(* IEC 61131-3 sources: generating_plc_code_with_llms/Code#2/ChatGPT_3.5/third run, 21 files *)

(* ---- 14.st ---- *)
// 7.98s
// 2
FUNCTION FC1001 : BOOL
VAR_INPUT
	MEW: REAL;
	SP: REAL;
	HYS: REAL;
END_VAR

VAR_IN_OUT
 	OUT: BOOL;
END_VAR

VAR
 	P_HYS: REAL;
END_VAR

// Calculate the switching hysteresis value
P_HYS := SP * (HYS / 100.0);

// Switch on if the measured value exceeds the setpoint + hysteresis
IF MEW > (SP + P_HYS) THEN
    OUT := TRUE;
END_IF;

// Switch off if the measured value falls below the setpoint - hysteresis
IF MEW < (SP - P_HYS) THEN
    OUT := FALSE;
END_IF;

// Return the output state
RETURN OUT;

END_FUNCTION

(* ---- 15.st ---- *)
// 11.59s
// 2
FUNCTION FC1002 : BOOL
VAR_INPUT
	E_A, SENSOR: BOOL;
	ZEITW: TIME;
END_VAR

VAR_IN_OUT
	ZEIT: TON;
	P_HU, P_AL: BOOL;
END_VAR

// Check if the monitoring system is switched on
IF E_A THEN
    // Check if the ultrasonic sensor detects an approach
    IF SENSOR THEN
        // Start the timer if it's not running
        IF NOT ZEIT.IN THEN
            ZEIT(IN := TRUE, PT := ZEITW);
        ELSE
            // Check if the timer has reached the set time
            IF ZEIT.Q THEN
                // Turn off the warning signal and switch on the alarm
                P_HU := FALSE;
                P_AL := TRUE;
            END_IF;
        END_IF;
    ELSE
        // Reset the timer if no approach is detected
        ZEIT(IN := FALSE);
    END_IF;

    // Check if the timer is not running
    IF NOT ZEIT.IN THEN
        // Check if the alarm is active and turn it off
        IF P_AL THEN
            P_AL := FALSE;
        END_IF;

        // Turn on the warning signal if an approach is detected
        P_HU := SENSOR;
    END_IF;
ELSE
    // Turn off both the warning signal and the alarm if the monitoring system is switched off
    P_HU := FALSE;
    P_AL := FALSE;
    // Reset the timer
    ZEIT(IN := FALSE);
END_IF;

// Return the output state
RETURN E_A;

END_FUNCTION

(* ---- 18.st ---- *)
// 8.25s
// 4
FUNCTION FC1003 : VOID
VAR_INPUT
    IN_R:REAL;
    IN_MAX, IN_MIN:REAL;
    OUT_MAX, OUT_MIN:REAL;
END_VAR
VAR_OUTPUT
    OUT_R:REAL;
    FEH:BOOL;
END_VAR
VAR_TEMP
    DIFF1, DIFF2:REAL;
END_VAR

IF IN_MAX <> IN_MIN AND OUT_MAX <> OUT_MIN THEN
    // Calculate the difference between input and output ranges
    DIFF1 := IN_MAX - IN_MIN;
    DIFF2 := OUT_MAX - OUT_MIN;

    // Check if the input value is within the specified range
    IF IN_R >= IN_MIN AND IN_R <= IN_MAX THEN
        // Map the input value to the output range
        OUT_R := ((IN_R - IN_MIN) / DIFF1) * DIFF2 + OUT_MIN;
        FEH := FALSE;
    ELSE
        // Input value is out of range
        OUT_R := 0.0;
        FEH := TRUE;
    END_IF;
ELSE
    // Invalid range configuration
    OUT_R := 0.0;
    FEH := TRUE;
END_IF;

(* ---- 19.st ---- *)
// 11.08s
// 2
FUNCTION_BLOCK FB1005
VAR_INPUT
    START: BOOL;
    DICKE, V_MAX, V_MIN: REAL;
END_VAR

VAR_OUTPUT
    D_MAX, D_MIN: REAL;
    P1: BOOL;
END_VAR

VAR
    FO: BOOL;
    OldDicke: REAL;
END_VAR

METHOD MeasureThickness: BOOL
    VAR
        Messwert: REAL;
    END_VAR
    // Measurement logic goes here
    // Replace the following line with your actual measurement code
    Messwert := ABS(RAND(1.0));
    D_MAX := MAX(Messwert, D_MAX);
    D_MIN := MIN(Messwert, D_MIN);
    RETURN TRUE;
END_METHOD

METHOD CheckReject: BOOL
    // Check if the measured values are outside the tolerance band
    IF (D_MAX > V_MAX OR D_MIN < V_MIN) THEN
        P1 := TRUE; // Switch on reject light
        RETURN TRUE;
    ELSE
        P1 := FALSE; // Switch off reject light
        RETURN FALSE;
    END_IF;
END_METHOD

METHOD ResetValues: BOOL
    // Reset measured values at the start of a new measurement cycle
    D_MAX := 0.0;
    D_MIN := 9999.9; // Adjust the initial value based on your actual expected range
    RETURN TRUE;
END_METHOD

METHOD FBExecution: BOOL
    // Main execution logic of the function block
    IF START THEN
        IF NOT FO THEN
            // Start a new measurement cycle
            ResetValues();
            FO := TRUE;
        END_IF;

        // Perform thickness measurement
        IF MeasureThickness() THEN
            // Check for reject condition
            CheckReject();
        END_IF;
    ELSE
        FO := FALSE; // Reset the flag when the sensor signal is not active
    END_IF;

    RETURN TRUE;
END_METHOD

END_FUNCTION_BLOCK

(* ---- 20.st ---- *)
// 10.41s
// 4
FUNCTION_BLOCK INTERLOCK
    VAR_INPUT
        I1 : BOOL;
        I2 : BOOL;
        TL : TIME;
    END_VAR

    VAR_OUTPUT
        Q1 : BOOL;
        Q2 : BOOL;
    END_VAR

    VAR
        T1 : TOF;
        T2 : TOF;
    END_VAR

    // Interlock logic
    T1(IN := I1 AND NOT Q2, PT := TL);
    T2(IN := I2 AND NOT Q1, PT := TL);

    Q1 := I1 AND NOT T2.Q;
    Q2 := I2 AND NOT T1.Q;

END_FUNCTION_BLOCK

(* ---- 21.st ---- *)
// 36.26s
// 2
FUNCTION_BLOCK BURNER
VAR_INPUT
    IN : BOOL;
    STAGE2 : BOOL;
    OVER_TEMP : BOOL;
    OIL_TEMP : BOOL := TRUE;
    FLAME : BOOL;
    RST : BOOL;
    RST_TIMER : BOOL;
    PRE_HEAT_TIME : TIME := t#5s;
    PRE_VENT_TIME : TIME := t#15s;
    PRE_IGNITE_TIME : TIME := t#15s;
    POST_IGNITE_TIME : TIME := t#25s;
    STAGE2_DELAY : TIME := t#10s;
    SAFETY_TIME : TIME := t#5s;
    LOCKOUT_TIME : TIME := t#10s;
    MULTIPLE_IGNITION : BOOL := TRUE;
    KW1 : REAL;
    KW2 : REAL;
END_VAR
VAR_OUTPUT
    MOTOR : BOOL;
    COIL1 : BOOL;
    COIL2 : BOOL;
    PRE_HEAT : BOOL;
    IGNITE : BOOL;
    FAIL : BOOL;
    KWH : REAL;
    STATUS : BYTE;
END_VAR
VAR_IN_OUT
    RUNTIME1 : UDINT;
    RUNTIME2 : UDINT;
    CYCLES : UDINT;
END_VAR
VAR
    state : INT := 110; // Initial state: Standby
    last : TIME;
    tx : TIME;
    last_change : TIME;
    timer1 : TON;
    timer2 : TON;
    oil_temp_last : BOOL;
    cycles2 : UDINT;
END_VAR

METHOD RunBurner: BOOL
    // State Machine Logic
    CASE state OF
        110: // Standby
            IF IN AND NOT OVER_TEMP THEN
                state := 111; // Startup sequence
                last := TON_TIME();
            END_IF;
        111: // Startup sequence
            PRE_HEAT := TRUE;
            IF TON(TIME() - last, PRE_HEAT_TIME) THEN
                IF OIL_TEMP AND NOT FLAME THEN
                    last := TON_TIME();
                    state := 112; // Burner runs on stage 1
                    CYCLES := CYCLES + 1;
                    RUNTIME1 := RUNTIME1 + (TIME() - last_change);
                END_IF;
            END_IF;
        112: // Burner runs on stage 1
            MOTOR := TRUE;
            COIL1 := TRUE;
            COIL2 := FALSE;

            IF STAGE2 AND TON(TIME() - last_change, STAGE2_DELAY) THEN
                state := 113; // Burner runs at stage 2
                timer2.IN := FALSE; // Reset timer2
            END_IF;
        113: // Burner runs at stage 2
            MOTOR := TRUE;
            COIL1 := FALSE;
            COIL2 := TRUE;

            // Check for flame sensor response
            IF FLAME THEN
                timer2.IN := TRUE; // Start timer2
                IF timer2.Q THEN
                    STATUS := 5; // Flame stops in operation
                    FAIL := TRUE;
                END_IF;
            END_IF;

            // Check for multiple ignition
            IF FLAME AND MULTIPLE_IGNITION THEN
                IGNITE := TRUE;
                MULTIPLE_IGNITION := FALSE;
            END_IF;

            // Check for flame break
            IF NOT FLAME AND MULTIPLE_IGNITION THEN
                IGNITE := FALSE;
            END_IF;

            // Check for stage 2 activation
            IF STAGE2 AND NOT FLAME THEN
                state := 113; // Continue at stage 2
            END_IF;

            // Check for over temperature
            IF OVER_TEMP THEN
                STATUS := 9; // Boiler overheating contact has tripped
                FAIL := TRUE;
                state := 110; // Standby
            END_IF;

            // Check for lockout time
            IF RST_TIMER THEN
                timer1.IN := FALSE; // Reset timer1
                state := 110; // Standby
            END_IF;
    END_CASE;

    // Calculate KWH
    KWH := (REAL(CYCLES) * KW1 * TO_REAL(RUNTIME1) / 3600) + (REAL(cycles2) * KW2 * TO_REAL(RUNTIME2) / 3600);

    // Return true if the burner is active
    RETURN (state = 111 OR state = 112 OR state = 113);
END_METHOD;
END_FUNCTION_BLOCK

(* ---- 1.st ---- *)
// 5.64s
// 3
VAR
    xAllOn : BOOL;
    xAllOff : BOOL;

    xAlarm1 : BOOL;
    xAlarm2 : BOOL;
END_VAR

xAllOn := FALSE;  // Initializing the signals
xAllOff := FALSE;

// Set all alarms to TRUE and turn off the signal
IF xAllOn THEN
    xAlarm1 := TRUE;
    xAlarm2 := TRUE;
    xAllOn := FALSE;
END_IF

// Set all alarms to FALSE and turn off the signal
IF xAllOff THEN
    xAlarm1 := FALSE;
    xAlarm2 := FALSE;
    xAllOff := FALSE;
END_IF

(* ---- 10.st ---- *)
// 4.04s
// 4
VAR_INPUT
    X : REAL;
END_VAR

VAR
    sigmoidResult : REAL;
END_VAR

// Sigmoid function implementation
sigmoidResult := 1 / (1 + EXP(-X));

(* ---- 11.st ---- *)
// 4.57s
// 4
VAR_INPUT
    x : REAL;
END_VAR

VAR
    signResult : INT;
END_VAR

// Sign function implementation
IF x > 0 THEN
    signResult := 1;
ELSIF x < 0 THEN
    signResult := -1;
ELSE
    signResult := 0;
END_IF

(* ---- 12.st ---- *)
// 3.47s
// 4
VAR
    X : REAL;
    sinhResult : REAL;
END_VAR

// Hyperbolic sine function implementation
sinhResult := (EXP(X) - EXP(-X)) / 2.0;

(* ---- 13.st ---- *)
// 7.42s
// 2
VAR CONSTANT
    MAXNUMBERS : UINT := 99;
END_VAR

VAR
    aNumbers : ARRAY[0..MAXNUMBERS] OF INT;
    nCnt : INT;
END_VAR

// Initialize the array with random numbers (replace this with your logic)
FOR nCnt := 0 TO MAXNUMBERS DO
    aNumbers[nCnt] := SOME_RANDOM_NUMBER_FUNCTION();
END_FOR

// Search for the specific number (10) in the list
nCnt := 0;

REPEAT
    IF aNumbers[nCnt] = 10 THEN
        // Abort the search if the number 10 is found
        EXIT;
    END_IF

    nCnt := nCnt + 1;
UNTIL nCnt > MAXNUMBERS;

// Check if the number 10 was found or not
IF nCnt <= MAXNUMBERS THEN
    // Number 10 was found
    // Your logic for when the number is found
ELSE
    // Number 10 was not found
    // Your logic for when the number is not found
END_IF

(* ---- 16.st ---- *)
// 13.32s
// 2
VAR
    North_green : BOOL;
    North_yellow : BOOL;
    North_red : BOOL;
    East_green : BOOL;
    East_yellow : BOOL;
    East_red : BOOL;
    T1 : TON;
END_VAR

T1(IN:=TRUE, PT:=10000);

IF T1.Q THEN
    // Between 0ms and 5000ms, North is green, and East is red
    North_green := TRUE;
    North_yellow := FALSE;
    North_red := FALSE;
    East_green := FALSE;
    East_yellow := FALSE;
    East_red := TRUE;
ELSIF T1.ET < 5000 THEN
    // Between 5000ms and 5500ms, North turns yellow
    North_green := FALSE;
    North_yellow := TRUE;
    North_red := FALSE;
    East_green := FALSE;
    East_yellow := FALSE;
    East_red := TRUE;
ELSIF T1.ET < 9500 THEN
    // Between 5500ms and 9500ms, North is red, and East is green
    North_green := FALSE;
    North_yellow := FALSE;
    North_red := TRUE;
    East_green := TRUE;
    East_yellow := FALSE;
    East_red := FALSE;
ELSE
    // Between 9500ms and 10000ms, East turns yellow
    North_green := FALSE;
    North_yellow := FALSE;
    North_red := TRUE;
    East_green := FALSE;
    East_yellow := TRUE;
    East_red := FALSE;
END_IF;

(* ---- 17.st ---- *)
// 6.33s
// 4
VAR
    aiOutside : INT;
    aiHumidity : INT;
    sShowText : STRING[80];
END_VAR

// Assume aiOutside represents temperature and aiHumidity represents humidity

// Evaluate temperature
IF aiOutside < 18 THEN
    sShowText := 'Cold';
ELSIF aiOutside >= 18 AND aiOutside <= 25 THEN
    // Evaluate humidity for the "Opt" condition
    IF aiHumidity >= 40 AND aiHumidity <= 75 THEN
        sShowText := 'Opt';
    ELSE
        sShowText := 'Temp. OK';
    END_IF;
ELSE
    sShowText := 'Hot';
END_IF;

(* ---- 2.st ---- *)
// 4.04s
// 4
VAR_INPUT
    N : INT;
    K : INT;
    i : INT;
END_VAR

VAR
    result : INT;
END_VAR

result := 1;

// Calculate N choose K
FOR i := 1 TO K DO
    result := result * (N - i + 1) / i;
END_FOR

(* ---- 3.st ---- *)
// 5.38s
// 2
VAR_INPUT
    X : INT;
END_VAR

VAR
    t1 : DINT;
    t2 : DINT;
    x_tmp : INT;
END_VAR

t1 := 0;
t2 := 1;

// Calculate Fibonacci number
IF X = 0 THEN
    x_tmp := t1;
ELSIF X = 1 THEN
    x_tmp := t2;
ELSE
    FOR i := 2 TO X DO
        x_tmp := t1 + t2;
        t1 := t2;
        t2 := x_tmp;
    END_FOR
END_IF

(* ---- 4.st ---- *)
// 6.26s
// 2
VAR
    aiLevel : INT;
    PercentLevel : UINT;
    doLow : BOOL;
    doOk : BOOL;
    doHigh : BOOL;
    doAlarm : BOOL;
END_VAR

// Read analog input for fill level (0 - 32767)
aiLevel := ... // Read the actual analog input value from your sensor

// Convert to percentage
PercentLevel := UINT_TO((aiLevel * 100) / 32767);

// Initialize output variables
doLow := FALSE;
doOk := FALSE;
doHigh := FALSE;
doAlarm := FALSE;

// Check fill level ranges using CASE instruction
CASE PercentLevel OF
    0 TO 1:
        doLow := TRUE;
        doAlarm := TRUE;
    2 TO 70:
        doOk := TRUE;
    71 TO 100:
        doHigh := TRUE;
END_CASE

(* ---- 5.st ---- *)
// 7.71s
// 4
VAR
    Start_Loop : BOOL := FALSE;
    one_hour : TIME := T#1h;
    One_Hour_Timer : TON;
    Gate_Open : BOOL := FALSE;
    Close_Gate_Inst : BOOL := FALSE;
    Sensed_Car : BOOL := FALSE;
    Sensed_Car_Inst : BOOL := FALSE;
    Sensed_App : BOOL := FALSE;
    Mobile_Inst : BOOL := FALSE;
    Auth : STRING;
    my_defined_str : STRING := 'abcd';
END_VAR

// Start the one-hour timer when Start_Loop is FALSE
One_Hour_Timer(IN := NOT Start_Loop, PT := one_hour);

// Check if the timer has timed out
IF One_Hour_Timer.Q THEN
    Close_Gate_Inst := TRUE;
    One_Hour_Timer(IN := FALSE); // Reset the timer
END_IF

// Check conditions to open the gate
IF (Sensed_Car AND Sensed_Car_Inst) OR (Sensed_App AND Mobile_Inst AND Auth = my_defined_str) THEN
    Gate_Open := TRUE;
    Close_Gate_Inst := FALSE; // Cancel closing the gate if it's open
END_IF

// Close the gate if required
IF Close_Gate_Inst THEN
    Gate_Open := FALSE;
END_IF

(* ---- 6.st ---- *)
// 13.35s
// 3
VAR CONSTANT
    WAIT : UINT := 0;
    TOP_POSITION : UINT := 1;
    BOTTOM_POSITION : UINT := 2;
    GETBOX : UINT := 3;
    UNLOAD_POSITION : UINT := 4;
    UNLOAD_BOX : UINT := 5;
END_VAR

VAR
    (*-- digital outputs*)
    doConvTop: BOOL;
    doConvBottom: BOOL;
    doConvLift: BOOL;
    doLiftTop: BOOL;
    doLiftBottom: BOOL;
    doLiftUnload: BOOL;
    (*-- digital inputs*)
    diConvTop: BOOL;
    diConvBottom: BOOL;
    diLiftTop: BOOL;
    diLiftBottom: BOOL;
    diLiftUnload: BOOL;
    diBoxLift: BOOL;
    (*-- status variables*)
    selectLift: UINT;
    ConvTopOn: BOOL;
    ConvBottomOn: BOOL;
END_VAR

CASE selectLift OF
    WAIT:
        // Wait for a conveyor belt to be activated
        IF diConvTop THEN
            doConvTop := FALSE; // Stop conveyor belt
            ConvTopOn := FALSE;
            selectLift := TOP_POSITION;
        ELSIF diConvBottom THEN
            doConvBottom := FALSE; // Stop conveyor belt
            ConvBottomOn := FALSE;
            selectLift := BOTTOM_POSITION;
        END_IF

    TOP_POSITION:
        // Move lift to top position
        IF NOT ConvTopOn THEN
            doLiftTop := TRUE;
            doLiftBottom := FALSE;
            ConvTopOn := TRUE;
        END_IF

        // Check if the lift is in the requested position
        IF diLiftTop THEN
            selectLift := GETBOX;
        END_IF

    BOTTOM_POSITION:
        // Move lift to bottom position
        IF NOT ConvBottomOn THEN
            doLiftTop := FALSE;
            doLiftBottom := TRUE;
            ConvBottomOn := TRUE;
        END_IF

        // Check if the lift is in the requested position
        IF diLiftBottom THEN
            selectLift := GETBOX;
        END_IF

    GETBOX:
        // Move the box onto the lift conveyor
        doConvLift := TRUE;

        // Check if the box is completely at the lift
        IF diBoxLift THEN
            doConvLift := FALSE; // Stop lift conveyor
            selectLift := UNLOAD_POSITION;
        END_IF

    UNLOAD_POSITION:
        // Move lift to unload position
        doLiftUnload := TRUE;

        // Check if the lift is in the unload position
        IF diLiftUnload THEN
            selectLift := UNLOAD_BOX;
        END_IF

    UNLOAD_BOX:
        // Move the box onto the unloading conveyor
        doConvLift := TRUE;

        // Check if the box has left the lift
        IF NOT diBoxLift THEN
            doConvLift := FALSE; // Stop lift conveyor
            selectLift := WAIT; // Reset for the next request
        END_IF
END_CASE

(* ---- 7.st ---- *)
// 7.3s
// 2
VAR CONSTANT
    MAX_INDEX: USINT := 4;
END_VAR

VAR
    aWeights : ARRAY[0..MAX_INDEX] OF INT;
    iCnt : USINT;
    sumWeight : DINT;
    avgWeight : INT;
END_VAR

// Initialize array with example values
aWeights := [10000, 8000, 12000, 6000, 9000];

// Calculate total load using a FOR loop
sumWeight := 0;
FOR iCnt := 0 TO MAX_INDEX DO
    sumWeight := sumWeight + aWeights[iCnt];
END_FOR

// Calculate average load
IF MAX_INDEX > 0 THEN
    avgWeight := sumWeight / (MAX_INDEX + 1);
ELSE
    avgWeight := 0;
END_IF

(* ---- 8.st ---- *)
// 7.13s
// 3
VAR_INPUT
    X : REAL;
END_VAR

VAR
    w : REAL;
    i : INT;
    we : REAL;
    w1e : REAL;
    ewx : REAL;
    last : DWORD;
END_VAR

// Initialize variables
w := 0.0;
last := 0;

FOR i := 1 TO 50 DO
    we := w * EXP(w);
    w1e := (w + 1.0) * EXP(w);
    ewx := EXP(w * X);

    w := w - (we - X) / (we + w1e - 2.0 * X * w1e / (2.0 * w + 1.0));

    IF ABS(last - REAL_TO_DWORD(w)) < 1 THEN
        EXIT;
    END_IF

    last := REAL_TO_DWORD(w);
END_FOR

(* ---- 9.st ---- *)
// 4.98s
// 2
VAR
    YEAR : INT;
END_VAR

// Check if the year is a leap year
IF (YEAR MOD 4 = 0 AND YEAR MOD 100 <> 0) OR (YEAR MOD 400 = 0) THEN
    // The year is a leap year
    // You can add your logic here for leap year
ELSE
    // The year is not a leap year
    // You can add your logic here for non-leap year
END_IF
